(* Schneider Machine Expert - Basic project resolucao, file version 2.7.0.0 *)
(* ProjectInformations: Name=Novo projeto *)

HARDWARE
  Cpu 0: TM221CE24R
  EthernetConfiguration: NetworkName=M221, IpAllocationMode=FixedAddress, IpAddress=0.0.0.0, SubnetMask=0.0.0.0
  SerialLineConfiguration: Baud=Baud19200, Parity=ParityEven, DataBits=DataBits8, StopBits=StopBits1, PhysicalMedium=PhysicalMediumRs485, TransmissionMode=TransmissionModeModbusRtu, SlaveId=1, Addressing=SlaveAddressing
  MastTask: UsePeriodScanMode=false, PeriodScan=100
  FastTask: Period=255
  CpuBehavior: StartingMode=StartAsPreviousState, AutoSaveRamOnEeprom=true, WatchdogPeriod=250

SYMBOLS  (address, symbol, comment, settings)
  %M0       SIG_IN_L1_ATU
  %M1       SIG_IN_L1_DESA
  %M2       SIG_IN_L2_ATU
  %M3       SIG_IN_L2_DESA
  %M4       SIG_IN_D1_ATU
  %M5       SIG_IN_D1_DESA
  %M6       SIG_IN_D2_ATU
  %M7       SIG_IN_D2_DESA
  %M20      SIG_RELE_R1_LIGA
  %M21      SIG_RELE_R1_DESL
  %M22      SIG_RELE_R2_LIGA
  %M23      SIG_RELE_R2_DESL
  %I0.1     IN_L1_ATU
  %I0.2     IN_L1_DESA
  %I0.3     IN_L2_ATU
  %I0.4     IN_L2_DESA
  %I0.5     IN_D1_ATU
  %I0.6     IN_D1_DESA
  %I0.7     IN_D2_ATU
  %I0.8     IN_D2_DESA
  %Q0.1     OUT_RELE_R1
  %Q0.2     OUT_RELE_R2

POU Entradas
  (* SectionNumber=1 *)

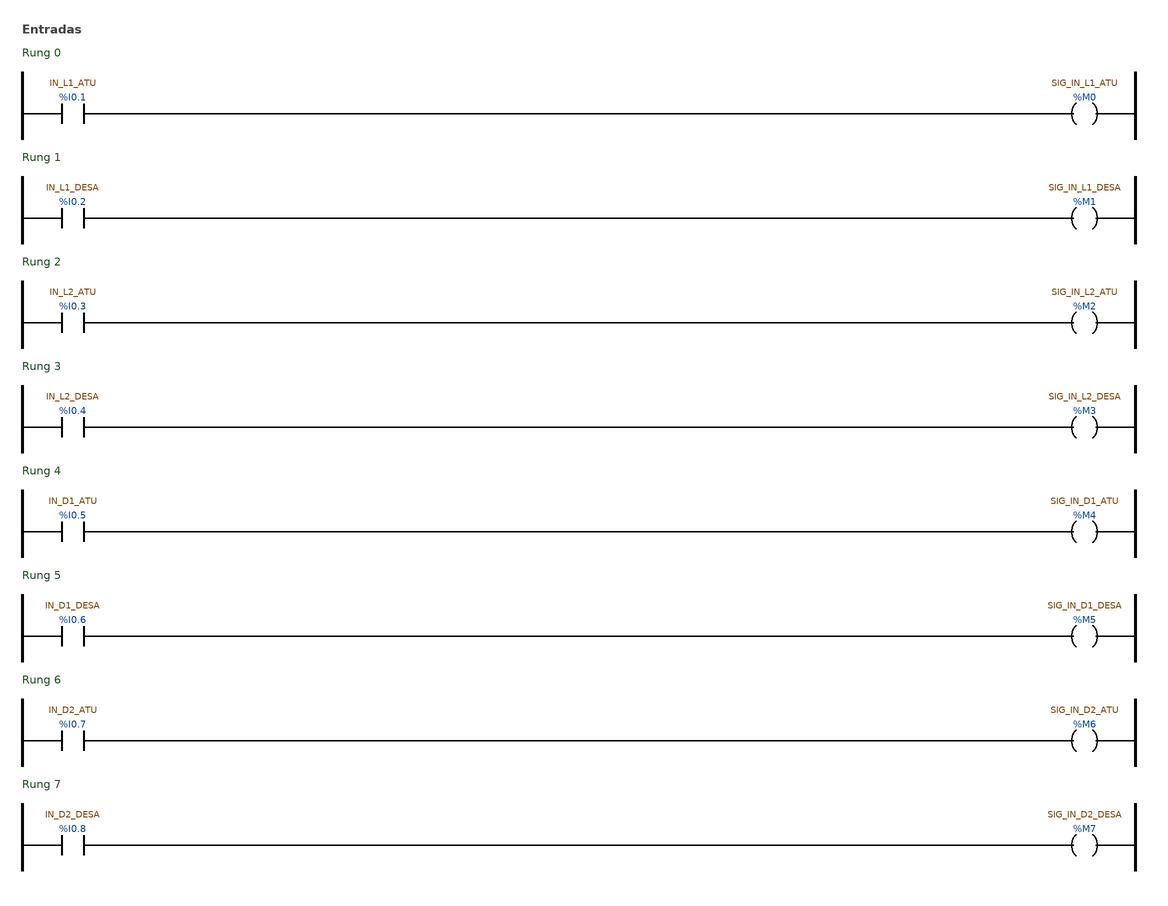

// Rung 0
  LD %I0.1                (* IN_L1_ATU *)
  ST %M0                  (* SIG_IN_L1_ATU *)
  // as ST:
  //   SIG_IN_L1_ATU := IN_L1_ATU;

// Rung 1
  LD %I0.2                (* IN_L1_DESA *)
  ST %M1                  (* SIG_IN_L1_DESA *)
  // as ST:
  //   SIG_IN_L1_DESA := IN_L1_DESA;

// Rung 2
  LD %I0.3                (* IN_L2_ATU *)
  ST %M2                  (* SIG_IN_L2_ATU *)
  // as ST:
  //   SIG_IN_L2_ATU := IN_L2_ATU;

// Rung 3
  LD %I0.4                (* IN_L2_DESA *)
  ST %M3                  (* SIG_IN_L2_DESA *)
  // as ST:
  //   SIG_IN_L2_DESA := IN_L2_DESA;

// Rung 4
  LD %I0.5                (* IN_D1_ATU *)
  ST %M4                  (* SIG_IN_D1_ATU *)
  // as ST:
  //   SIG_IN_D1_ATU := IN_D1_ATU;

// Rung 5
  LD %I0.6                (* IN_D1_DESA *)
  ST %M5                  (* SIG_IN_D1_DESA *)
  // as ST:
  //   SIG_IN_D1_DESA := IN_D1_DESA;

// Rung 6
  LD %I0.7                (* IN_D2_ATU *)
  ST %M6                  (* SIG_IN_D2_ATU *)
  // as ST:
  //   SIG_IN_D2_ATU := IN_D2_ATU;

// Rung 7
  LD %I0.8                (* IN_D2_DESA *)
  ST %M7                  (* SIG_IN_D2_DESA *)
  // as ST:
  //   SIG_IN_D2_DESA := IN_D2_DESA;

POU Lógicas
  (* SectionNumber=2 *)

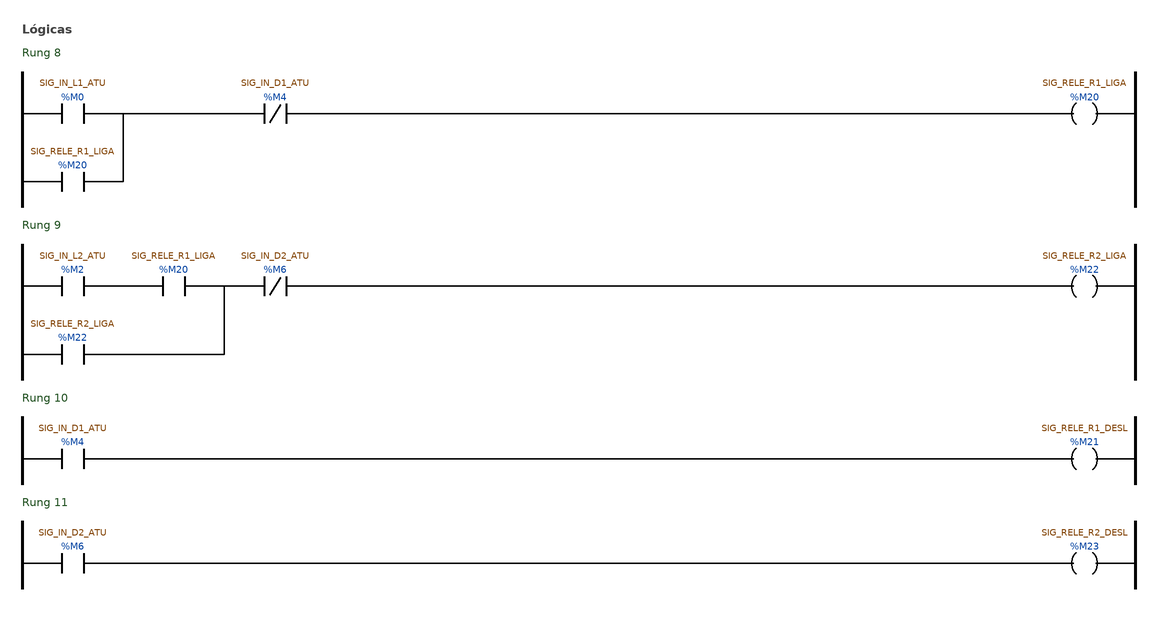

// Rung 8
  LD %M0                  (* SIG_IN_L1_ATU *)
  OR %M20                 (* SIG_RELE_R1_LIGA *)
  ANDN %M4                (* SIG_IN_D1_ATU *)
  ST %M20                 (* SIG_RELE_R1_LIGA *)
  // as ST:
  //   SIG_RELE_R1_LIGA := (SIG_IN_L1_ATU OR SIG_RELE_R1_LIGA) AND NOT SIG_IN_D1_ATU;

// Rung 9
  LD %M2                  (* SIG_IN_L2_ATU *)
  AND %M20                (* SIG_RELE_R1_LIGA *)
  OR %M22                 (* SIG_RELE_R2_LIGA *)
  ANDN %M6                (* SIG_IN_D2_ATU *)
  ST %M22                 (* SIG_RELE_R2_LIGA *)
  // as ST:
  //   SIG_RELE_R2_LIGA := (SIG_IN_L2_ATU AND SIG_RELE_R1_LIGA OR SIG_RELE_R2_LIGA) AND NOT SIG_IN_D2_ATU;

// Rung 10
  LD %M4                  (* SIG_IN_D1_ATU *)
  ST %M21                 (* SIG_RELE_R1_DESL *)
  // as ST:
  //   SIG_RELE_R1_DESL := SIG_IN_D1_ATU;

// Rung 11
  LD %M6                  (* SIG_IN_D2_ATU *)
  ST %M23                 (* SIG_RELE_R2_DESL *)
  // as ST:
  //   SIG_RELE_R2_DESL := SIG_IN_D2_ATU;

POU Saídas
  (* SectionNumber=3 *)

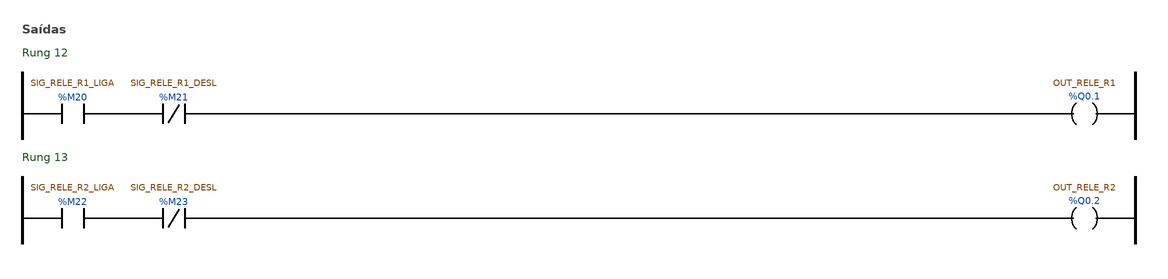

// Rung 12
  LD %M20                 (* SIG_RELE_R1_LIGA *)
  ANDN %M21               (* SIG_RELE_R1_DESL *)
  ST %Q0.1                (* OUT_RELE_R1 *)
  // as ST:
  //   OUT_RELE_R1 := SIG_RELE_R1_LIGA AND NOT SIG_RELE_R1_DESL;

// Rung 13
  LD %M22                 (* SIG_RELE_R2_LIGA *)
  ANDN %M23               (* SIG_RELE_R2_DESL *)
  ST %Q0.2                (* OUT_RELE_R2 *)
  // as ST:
  //   OUT_RELE_R2 := SIG_RELE_R2_LIGA AND NOT SIG_RELE_R2_DESL;
